PROGRAM GCC2
VAR
END_VAR

END_PROGRAM

(* stored: Version 1.1.0.1, ProductVersion 3.1.4022.3
   POU GCC2: Id {cd1af1d4-04a6-41fb-a0c2-978ed45d40cc}, SpecialFunc None *)
